// TIA Portal project "BTL_PLC_192" (V15)

(* hardware
DEVICE "S7300/ET200M station_1"  S7-300 station
   slot 0: "Rail_0"  Rail  6ES7 390-1***0-0AA0
   slot 2: "PLC_1"  CPU 314C-2 PN/DP  6ES7 314-6EH04-0AB0  V3.3
      slot 2: "PROFINET interface_1"  PN-IO
         slot 1: "Port_1"  Port
         slot 2: "Port_2"  Port
      slot 5: "DI 24/DO 16_1"  DI24/DO16
      slot 6: "AI 5/AO 2_1"  AI5/AO2
      slot 7: "Count_1"  Counter
      slot 8: "Positioning_1"  Positioning
*)

// ===== PLC "PLC_1"  CPU 314C-2 PN/DP =====

VAR_GLOBAL   // PLC tag table "Default tag table"
   "BI_AUTO" AT %I0.0 : Bool;
   "BI_MANU" AT %I0.1 : Bool;
   "BI_START" AT %I0.2 : Bool;
   "BI_STOP" AT %I0.3 : Bool;
   "I_CT1" AT %I0.4 : Bool;
   "I_CT2" AT %I0.5 : Bool;
   "I_CT3" AT %I0.6 : Bool;
   "I_CT4" AT %I0.7 : Bool;
   "IW_NHIET_DO" AT %IW64 : Int;
   "IW_ANH_SANG" AT %IW66 : Int;
   "IW_DO_AM" AT %IW68 : Int;
   "IW_DO_AM_DAT" AT %IW70 : Int;
   "BM_AUTO" AT %M0.0 : Bool;
   "BM_MANU" AT %M0.1 : Bool;
   "BM_START" AT %M0.2 : Bool;
   "BM_STOP" AT %M0.3 : Bool;
   "M_CT1" AT %M0.4 : Bool;
   "M_CT2" AT %M0.5 : Bool;
   "M_CT3" AT %M0.6 : Bool;
   "M_CT4" AT %M0.7 : Bool;
   "MW_NHIET_DO" AT %MW64 : Int;
   "MW_ANH_SANG" AT %MW66 : Int;
   "MW_DO_AM" AT %MW68 : Int;
   "MW_DO_AM_DAT" AT %MW70 : Int;
   "BM_SIMULATION" AT %M1.0 : Bool;
   "BIT_GIU" AT %M1.1 : Bool;
   "BIT_TUOI_THEO_TIME_THUC" AT %M1.2 : Bool;
   "BIT_TUOI_THEO_ND" AT %M1.3 : Bool;
   "BIT_TUOI_THEO_DA" AT %M1.4 : Bool;
   "BIT_TUOI_THEO_DAD" AT %M1.5 : Bool;
   "Q_DEN_LV" AT %Q0.0 : Bool;
   "Q_QTG1" AT %Q0.1 : Bool;
   "Q_QTG2" AT %Q0.2 : Bool;
   "Q_BPS" AT %Q0.3 : Bool;
   "Q_GN1" AT %Q0.4 : Bool;
   "Q_GN2" AT %Q0.5 : Bool;
   "Q_MC_CLOSE" AT %Q0.6 : Bool;
   "Q_MC_OPEN" AT %Q0.7 : Bool;
   "Q_BNV" AT %Q1.0 : Bool;
   "Q_QHA1" AT %Q1.1 : Bool;
   "Q_QHA2" AT %Q1.2 : Bool;
   "Q_DCS" AT %Q1.3 : Bool;
   "Auto" AT %M1.6 : Bool;
   "Manu" AT %M1.7 : Bool;
   "AUTO_RUN" AT %M2.0 : Bool;
   "MANU_RUN" AT %M2.1 : Bool;
   "SIM_MODE" AT %M2.2 : Bool;
   "RET_VAL1" AT %MW4 : Word;
   "BIPOLAR" AT %M2.3 : Bool;
   "RET_VAL2" AT %MW6 : Word;
   "RET_VAL3" AT %MW8 : Word;
   "RET_VAL4" AT %MW10 : Word;
   "RET_VAL5" AT %MW12 : Int;
   "ALWAY_OFF" AT %M2.4 : Bool;
   "TT_DATE_OF_WEEK" AT %MW194 : Int;
   "Tag_M" AT %M2.6 : Bool;
   "Tag_M1" AT %M2.7 : Bool;
   "TIME_TUOI" AT %MW14 : Int;
   "tag_M3" AT %M2.5 : Bool;
   "tag_M4" AT %M3.0 : Bool;
   "Tag_M5" AT %M3.1 : Bool;
   "Tag_M6" AT %M3.2 : Bool;
   "Tag_M7" AT %M3.3 : Bool;
   "Tag_M8" AT %M3.4 : Bool;
   "Tag_M9" AT %M3.5 : Bool;
   "Tag_1" AT %T1 : Timer;
END_VAR

VAR_GLOBAL   // PLC tag table "Tag table_1"
   "TT_NHIET_DO" AT %MD100 : Real;
   "TT_ANH_SANG" AT %MD104 : Real;
   "TT_DO_AM" AT %MD108 : Real;
   "SET_MAX_ND" AT %MD112 : Real;
   "SET_MIN_ND" AT %MD116 : Real;
   "SET_MAX_AS" AT %MD120 : Real;
   "SET_MIN_AS" AT %MD124 : Real;
   "SET_MAX_DO_AM" AT %MD128 : Real;
   "SET_MIN_DO_AM" AT %MD132 : Real;
   "SET_NGAY1" AT %MW148 : Int;
   "SET_GIO1" AT %MW150 : Int;
   "SET_PHUT1" AT %MW152 : Int;
   "TT_NGAY" AT %MW154 : Int;
   "TT_GIO" AT %MW156 : Int;
   "TT_PHUT" AT %MW158 : Int;
   "TT_GIAY" AT %MW160 : Int;
   "TT_NAM" AT %MW162 : Int;
   "TT_THANG" AT %MW164 : Int;
   "SET_NGAY2" AT %MW166 : Int;
   "SET_GIO2" AT %MW168 : Int;
   "SET_PHUT2" AT %MW170 : Int;
   "SET_NGAY3" AT %MW172 : Int;
   "SET_GIO3" AT %MW174 : Int;
   "SET_PHUT3" AT %MW176 : Int;
   "SET_TIME_TUOI" AT %MW178 : Int;
   "SET_MAX_DO_AM_DAT" AT %MD200 : Real;
   "SET_MIN_DO_AM_DAT" AT %MD204 : Real;
   "TT_DO_AM_DAT" AT %MD208 : Real;
   "TT_TIME_TUOI" AT %MW214 : Int;
   "SET_NHIET_DO" AT %MD216 : Real;
   "SET_DAD" AT %MD220 : Real;
   "SET_DO_AM_KK" AT %MD224 : Real;
   "SET_ANH_SANG" AT %MD228 : Real;
END_VAR

VAR_GLOBAL   // PLC tag table "Tag table_2"
   "START_BPS" AT %M20.0 : Bool;
   "STOP_BPS" AT %M20.1 : Bool;
   "START_QTG" AT %M20.2 : Bool;
   "STOP_QTG" AT %M20.3 : Bool;
   "START_DEN_CHIEU_SANG" AT %M20.4 : Bool;
   "STOP_DEN_CHIEU_SANG" AT %M20.5 : Bool;
   "START_QUAT_HUT_AM" AT %M20.6 : Bool;
   "STOP_QUAT_HUT_AM" AT %M20.7 : Bool;
   "START_GN" AT %M21.0 : Bool;
   "STOP_GN" AT %M21.1 : Bool;
   "OPEN_MAI_CHE" AT %M21.2 : Bool;
   "CLOSE_MAI_CHE" AT %M21.3 : Bool;
END_VAR

FUNCTION "MAY BOM SUONG" : Void   // FC1, LAD
{ S7_Optimized_Access := 'FALSE' }
VERSION : 0.1
   VAR_INPUT
      SET_GIO1 : Int;
      SET_PHUT1 : Int;
      SET_GIO2 : Int;
      SET_PHUT2 : Int;
      SET_GIO3 : Int;
      SET_PHUT3 : Int;
   END_VAR
   VAR_OUTPUT
      MAY_BOM_PS : Bool;
      GIA_NHIET1 : Bool;
      GIA_NHIET2 : Bool;
      QUAT_TG1 : Bool;
      QUAT_TG2 : Bool;
      QUAT_HUT_AM1 : Bool;
      QUAT_HUT_AM2 : Bool;
      BOM_NUOC_TANK : Bool;
   END_VAR
   VAR_TEMP
      ALWAYS_OFF : Bool;
      temp : Bool;
      LOOP : Bool;
      temp2 : Bool;
      TT_TUOI : Int;
   END_VAR
   VAR_TEMP   // added for the SCL form of the ladder/FBD networks
      _w1 : Bool;
   END_VAR
BEGIN

REGION Network 1: Đặt thời gian tưới trong ngày( tưới 3 lần 1 ngày)
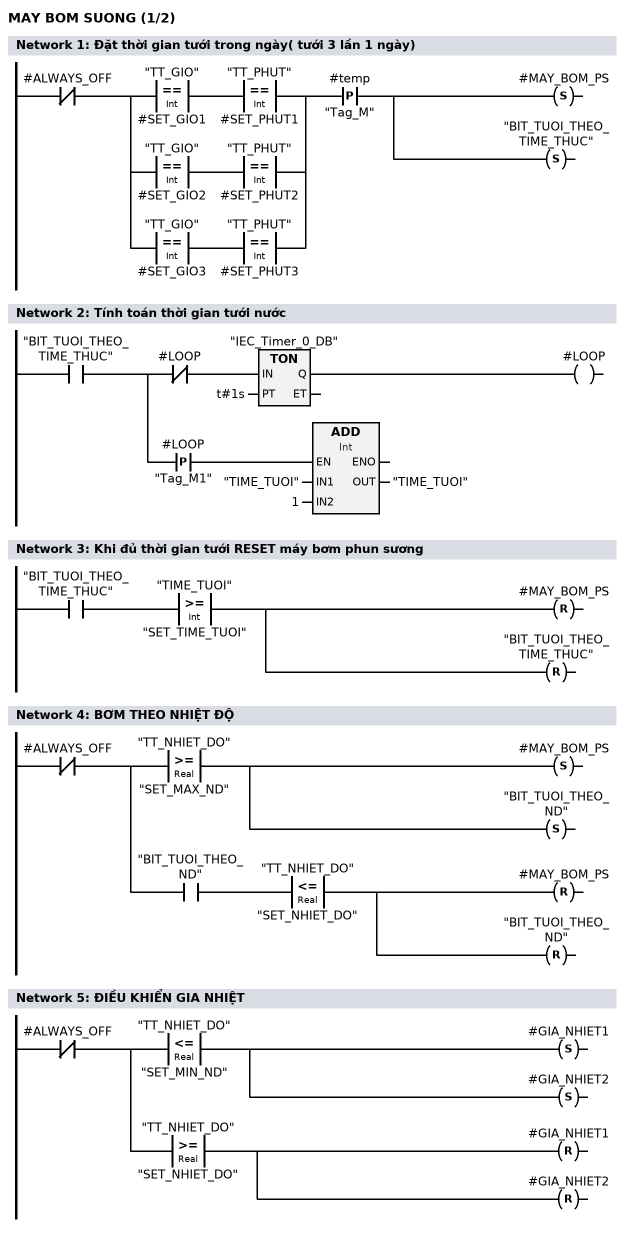
   RUNG wire#powerrail
      I_Contact( #ALWAYS_OFF )
      wire#w1
      { S7_Templates := "SrcType := Int" } EQ_Contact(in1 := "TT_GIO", in2 := #SET_GIO1)
      { S7_Templates := "SrcType := Int" } EQ_Contact(in1 := "TT_PHUT", in2 := #SET_PHUT1)
      wire#w2
      P_Contact(operand := #temp, bit := "Tag_M")
      wire#w3
      S_Coil( #MAY_BOM_PS )
   END_RUNG
   RUNG wire#w1
      { S7_Templates := "SrcType := Int" } EQ_Contact(in1 := "TT_GIO", in2 := #SET_GIO2)
      { S7_Templates := "SrcType := Int" } EQ_Contact(in1 := "TT_PHUT", in2 := #SET_PHUT2)
   END_RUNG wire#w2
   RUNG wire#w1
      { S7_Templates := "SrcType := Int" } EQ_Contact(in1 := "TT_GIO", in2 := #SET_GIO3)
      { S7_Templates := "SrcType := Int" } EQ_Contact(in1 := "TT_PHUT", in2 := #SET_PHUT3)
   END_RUNG wire#w2
   RUNG wire#w3
      S_Coil( "BIT_TUOI_THEO_TIME_THUC" )
   END_RUNG
   // the same network as SCL:
   #_w1 := NOT #ALWAYS_OFF AND ((("TT_GIO" = #SET_GIO1) AND ("TT_PHUT" = #SET_PHUT1)) OR (("TT_GIO" = #SET_GIO2) AND ("TT_PHUT" = #SET_PHUT2)) OR (("TT_GIO" = #SET_GIO3) AND ("TT_PHUT" = #SET_PHUT3))) AND #temp AND NOT "Tag_M";   // rising edge of #temp
   "Tag_M" := #temp;
   IF #_w1 THEN
       #MAY_BOM_PS := TRUE;
       "BIT_TUOI_THEO_TIME_THUC" := TRUE;
   END_IF;
END_REGION

REGION Network 2: Tính toán thời gian tưới nước
   "IEC_Timer_0_DB".TON(IN := "BIT_TUOI_THEO_TIME_THUC" AND NOT #LOOP, PT := t#1s);
   #LOOP := "IEC_Timer_0_DB".Q;
   #_w1 := "BIT_TUOI_THEO_TIME_THUC" AND #LOOP AND NOT "Tag_M1";   // rising edge of #LOOP
   "Tag_M1" := #LOOP;
   IF #_w1 THEN "TIME_TUOI" := "TIME_TUOI" + 1; END_IF;
END_REGION

REGION Network 3: Khi đủ thời gian tưới RESET máy bơm phun sương
   RUNG wire#powerrail
      Contact( "BIT_TUOI_THEO_TIME_THUC" )
      { S7_Templates := "SrcType := Int" } GE_Contact(in1 := "TIME_TUOI", in2 := "SET_TIME_TUOI")
      wire#w1
      R_Coil( #MAY_BOM_PS )
   END_RUNG
   RUNG wire#w1
      R_Coil( "BIT_TUOI_THEO_TIME_THUC" )
   END_RUNG
   // the same network as SCL:
   IF "BIT_TUOI_THEO_TIME_THUC" AND ("TIME_TUOI" >= "SET_TIME_TUOI") THEN
       #MAY_BOM_PS := FALSE;
       "BIT_TUOI_THEO_TIME_THUC" := FALSE;
   END_IF;
END_REGION

REGION Network 4: BƠM THEO NHIỆT ĐỘ
   RUNG wire#powerrail
      I_Contact( #ALWAYS_OFF )
      wire#w1
      { S7_Templates := "SrcType := Real" } GE_Contact(in1 := "TT_NHIET_DO", in2 := "SET_MAX_ND")
      wire#w2
      S_Coil( #MAY_BOM_PS )
   END_RUNG
   RUNG wire#w2
      S_Coil( "BIT_TUOI_THEO_ND" )
   END_RUNG
   RUNG wire#w1
      Contact( "BIT_TUOI_THEO_ND" )
      { S7_Templates := "SrcType := Real" } LE_Contact(in1 := "TT_NHIET_DO", in2 := "SET_NHIET_DO")
      wire#w3
      R_Coil( #MAY_BOM_PS )
   END_RUNG
   RUNG wire#w3
      R_Coil( "BIT_TUOI_THEO_ND" )
   END_RUNG
   // the same network as SCL:
   IF NOT #ALWAYS_OFF AND ("TT_NHIET_DO" >= "SET_MAX_ND") THEN
       #MAY_BOM_PS := TRUE;
       "BIT_TUOI_THEO_ND" := TRUE;
   END_IF;
   IF NOT #ALWAYS_OFF AND "BIT_TUOI_THEO_ND" AND ("TT_NHIET_DO" <= "SET_NHIET_DO") THEN
       #MAY_BOM_PS := FALSE;
       "BIT_TUOI_THEO_ND" := FALSE;
   END_IF;
END_REGION

REGION Network 5: ĐIỀU KHIỂN GIA NHIỆT
   RUNG wire#powerrail
      I_Contact( #ALWAYS_OFF )
      wire#w1
      { S7_Templates := "SrcType := Real" } LE_Contact(in1 := "TT_NHIET_DO", in2 := "SET_MIN_ND")
      wire#w2
      S_Coil( #GIA_NHIET1 )
   END_RUNG
   RUNG wire#w2
      S_Coil( #GIA_NHIET2 )
   END_RUNG
   RUNG wire#w1
      { S7_Templates := "SrcType := Real" } GE_Contact(in1 := "TT_NHIET_DO", in2 := "SET_NHIET_DO")
      wire#w3
      R_Coil( #GIA_NHIET1 )
   END_RUNG
   RUNG wire#w3
      R_Coil( #GIA_NHIET2 )
   END_RUNG
   // the same network as SCL:
   IF NOT #ALWAYS_OFF AND ("TT_NHIET_DO" <= "SET_MIN_ND") THEN
       #GIA_NHIET1 := TRUE;
       #GIA_NHIET2 := TRUE;
   END_IF;
   IF NOT #ALWAYS_OFF AND ("TT_NHIET_DO" >= "SET_NHIET_DO") THEN
       #GIA_NHIET1 := FALSE;
       #GIA_NHIET2 := FALSE;
   END_IF;
END_REGION

REGION Network 6: ĐIỀU KHIỂN MÁY BƠM THEO ĐỘ ẨM ĐẤT
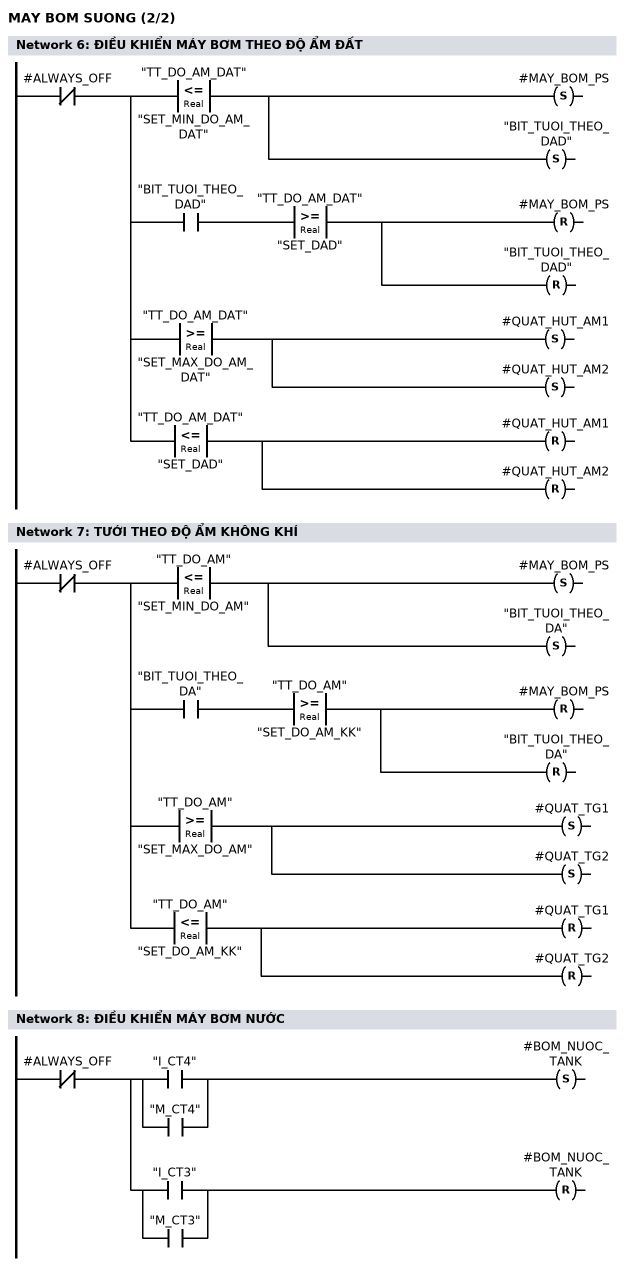
   RUNG wire#powerrail
      I_Contact( #ALWAYS_OFF )
      wire#w1
      { S7_Templates := "SrcType := Real" } LE_Contact(in1 := "TT_DO_AM_DAT", in2 := "SET_MIN_DO_AM_DAT")
      wire#w2
      S_Coil( #MAY_BOM_PS )
   END_RUNG
   RUNG wire#w2
      S_Coil( "BIT_TUOI_THEO_DAD" )
   END_RUNG
   RUNG wire#w1
      Contact( "BIT_TUOI_THEO_DAD" )
      { S7_Templates := "SrcType := Real" } GE_Contact(in1 := "TT_DO_AM_DAT", in2 := "SET_DAD")
      wire#w3
      R_Coil( #MAY_BOM_PS )
   END_RUNG
   RUNG wire#w3
      R_Coil( "BIT_TUOI_THEO_DAD" )
   END_RUNG
   RUNG wire#w1
      { S7_Templates := "SrcType := Real" } GE_Contact(in1 := "TT_DO_AM_DAT", in2 := "SET_MAX_DO_AM_DAT")
      wire#w4
      S_Coil( #QUAT_HUT_AM1 )
   END_RUNG
   RUNG wire#w4
      S_Coil( #QUAT_HUT_AM2 )
   END_RUNG
   RUNG wire#w1
      { S7_Templates := "SrcType := Real" } LE_Contact(in1 := "TT_DO_AM_DAT", in2 := "SET_DAD")
      wire#w5
      R_Coil( #QUAT_HUT_AM1 )
   END_RUNG
   RUNG wire#w5
      R_Coil( #QUAT_HUT_AM2 )
   END_RUNG
   // the same network as SCL:
   IF NOT #ALWAYS_OFF AND ("TT_DO_AM_DAT" <= "SET_MIN_DO_AM_DAT") THEN
       #MAY_BOM_PS := TRUE;
       "BIT_TUOI_THEO_DAD" := TRUE;
   END_IF;
   IF NOT #ALWAYS_OFF AND "BIT_TUOI_THEO_DAD" AND ("TT_DO_AM_DAT" >= "SET_DAD") THEN
       #MAY_BOM_PS := FALSE;
       "BIT_TUOI_THEO_DAD" := FALSE;
   END_IF;
   IF NOT #ALWAYS_OFF AND ("TT_DO_AM_DAT" >= "SET_MAX_DO_AM_DAT") THEN
       #QUAT_HUT_AM1 := TRUE;
       #QUAT_HUT_AM2 := TRUE;
   END_IF;
   IF NOT #ALWAYS_OFF AND ("TT_DO_AM_DAT" <= "SET_DAD") THEN
       #QUAT_HUT_AM1 := FALSE;
       #QUAT_HUT_AM2 := FALSE;
   END_IF;
END_REGION

REGION Network 7: TƯỚI THEO ĐỘ ẨM KHÔNG KHÍ
   RUNG wire#powerrail
      I_Contact( #ALWAYS_OFF )
      wire#w1
      { S7_Templates := "SrcType := Real" } LE_Contact(in1 := "TT_DO_AM", in2 := "SET_MIN_DO_AM")
      wire#w2
      S_Coil( #MAY_BOM_PS )
   END_RUNG
   RUNG wire#w2
      S_Coil( "BIT_TUOI_THEO_DA" )
   END_RUNG
   RUNG wire#w1
      Contact( "BIT_TUOI_THEO_DA" )
      { S7_Templates := "SrcType := Real" } GE_Contact(in1 := "TT_DO_AM", in2 := "SET_DO_AM_KK")
      wire#w3
      R_Coil( #MAY_BOM_PS )
   END_RUNG
   RUNG wire#w3
      R_Coil( "BIT_TUOI_THEO_DA" )
   END_RUNG
   RUNG wire#w1
      { S7_Templates := "SrcType := Real" } GE_Contact(in1 := "TT_DO_AM", in2 := "SET_MAX_DO_AM")
      wire#w4
      S_Coil( #QUAT_TG1 )
   END_RUNG
   RUNG wire#w4
      S_Coil( #QUAT_TG2 )
   END_RUNG
   RUNG wire#w1
      { S7_Templates := "SrcType := Real" } LE_Contact(in1 := "TT_DO_AM", in2 := "SET_DO_AM_KK")
      wire#w5
      R_Coil( #QUAT_TG1 )
   END_RUNG
   RUNG wire#w5
      R_Coil( #QUAT_TG2 )
   END_RUNG
   // the same network as SCL:
   IF NOT #ALWAYS_OFF AND ("TT_DO_AM" <= "SET_MIN_DO_AM") THEN
       #MAY_BOM_PS := TRUE;
       "BIT_TUOI_THEO_DA" := TRUE;
   END_IF;
   IF NOT #ALWAYS_OFF AND "BIT_TUOI_THEO_DA" AND ("TT_DO_AM" >= "SET_DO_AM_KK") THEN
       #MAY_BOM_PS := FALSE;
       "BIT_TUOI_THEO_DA" := FALSE;
   END_IF;
   IF NOT #ALWAYS_OFF AND ("TT_DO_AM" >= "SET_MAX_DO_AM") THEN
       #QUAT_TG1 := TRUE;
       #QUAT_TG2 := TRUE;
   END_IF;
   IF NOT #ALWAYS_OFF AND ("TT_DO_AM" <= "SET_DO_AM_KK") THEN
       #QUAT_TG1 := FALSE;
       #QUAT_TG2 := FALSE;
   END_IF;
END_REGION

REGION Network 8: ĐIỀU KHIỂN MÁY BƠM NƯỚC
   RUNG wire#powerrail
      I_Contact( #ALWAYS_OFF )
      wire#w1
      Contact( "I_CT4" )
      wire#w2
      S_Coil( #BOM_NUOC_TANK )
   END_RUNG
   RUNG wire#w1
      Contact( "M_CT4" )
   END_RUNG wire#w2
   RUNG wire#w1
      Contact( "I_CT3" )
      wire#w3
      R_Coil( #BOM_NUOC_TANK )
   END_RUNG
   RUNG wire#w1
      Contact( "M_CT3" )
   END_RUNG wire#w3
   // the same network as SCL:
   IF NOT #ALWAYS_OFF AND ("I_CT4" OR "M_CT4") THEN #BOM_NUOC_TANK := TRUE; END_IF;
   IF NOT #ALWAYS_OFF AND ("I_CT3" OR "M_CT3") THEN #BOM_NUOC_TANK := FALSE; END_IF;
END_REGION
END_FUNCTION

FUNCTION "MAI CHE" : Void   // FC2, LAD
{ S7_Optimized_Access := 'FALSE' }
VERSION : 0.1
   VAR_INPUT
      TT_ANH_SANG : Real;
      SET_MAX_AS : Real;
      SET_ANH_SANG : Real;
      SET_MIN_AS : Real;
   END_VAR
   VAR_OUTPUT
      MO_MAI_CHE : Bool;
      DEN_CHIEU_SANG : Bool;
      DONG_MAI_CHE : Bool;
   END_VAR
   VAR_TEMP
      ALWAYS_OFF : Bool;
   END_VAR
BEGIN

REGION Network 1
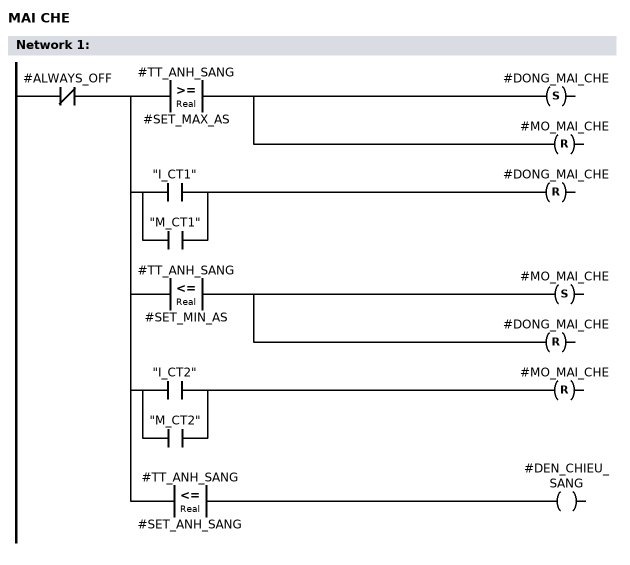
   RUNG wire#powerrail
      I_Contact( #ALWAYS_OFF )
      wire#w1
      { S7_Templates := "SrcType := Real" } GE_Contact(in1 := #TT_ANH_SANG, in2 := #SET_MAX_AS)
      wire#w2
      S_Coil( #DONG_MAI_CHE )
   END_RUNG
   RUNG wire#w2
      R_Coil( #MO_MAI_CHE )
   END_RUNG
   RUNG wire#w1
      Contact( "I_CT1" )
      wire#w3
      R_Coil( #DONG_MAI_CHE )
   END_RUNG
   RUNG wire#w1
      Contact( "M_CT1" )
   END_RUNG wire#w3
   RUNG wire#w1
      { S7_Templates := "SrcType := Real" } LE_Contact(in1 := #TT_ANH_SANG, in2 := #SET_MIN_AS)
      wire#w4
      S_Coil( #MO_MAI_CHE )
   END_RUNG
   RUNG wire#w4
      R_Coil( #DONG_MAI_CHE )
   END_RUNG
   RUNG wire#w1
      Contact( "I_CT2" )
      wire#w5
      R_Coil( #MO_MAI_CHE )
   END_RUNG
   RUNG wire#w1
      Contact( "M_CT2" )
   END_RUNG wire#w5
   RUNG wire#w1
      { S7_Templates := "SrcType := Real" } LE_Contact(in1 := #TT_ANH_SANG, in2 := #SET_ANH_SANG)
      Coil( #DEN_CHIEU_SANG )
   END_RUNG
   // the same network as SCL:
   IF NOT #ALWAYS_OFF AND (#TT_ANH_SANG >= #SET_MAX_AS) THEN
       #DONG_MAI_CHE := TRUE;
       #MO_MAI_CHE := FALSE;
   END_IF;
   IF NOT #ALWAYS_OFF AND ("I_CT1" OR "M_CT1") THEN #DONG_MAI_CHE := FALSE; END_IF;
   IF NOT #ALWAYS_OFF AND (#TT_ANH_SANG <= #SET_MIN_AS) THEN
       #MO_MAI_CHE := TRUE;
       #DONG_MAI_CHE := FALSE;
   END_IF;
   IF NOT #ALWAYS_OFF AND ("I_CT2" OR "M_CT2") THEN #MO_MAI_CHE := FALSE; END_IF;
   #DEN_CHIEU_SANG := NOT #ALWAYS_OFF AND (#TT_ANH_SANG <= #SET_ANH_SANG);
END_REGION
END_FUNCTION

FUNCTION "CHON CHE DO" : Void   // FC3, LAD
{ S7_Optimized_Access := 'FALSE' }
VERSION : 0.1
   VAR_INPUT
      S_AUTO : Bool;
      S_MANU : Bool;
      START : Bool;
      STOP : Bool;
   END_VAR
   VAR_OUTPUT
      MODE_AUTO : Bool;
      MODE_MANU : Bool;
   END_VAR
   VAR_TEMP
      AUTO : Bool;
      MANU : Bool;
   END_VAR
   VAR_TEMP   // added for the SCL form of the ladder/FBD networks
      _w1 : Bool;
   END_VAR
BEGIN

REGION Network 1
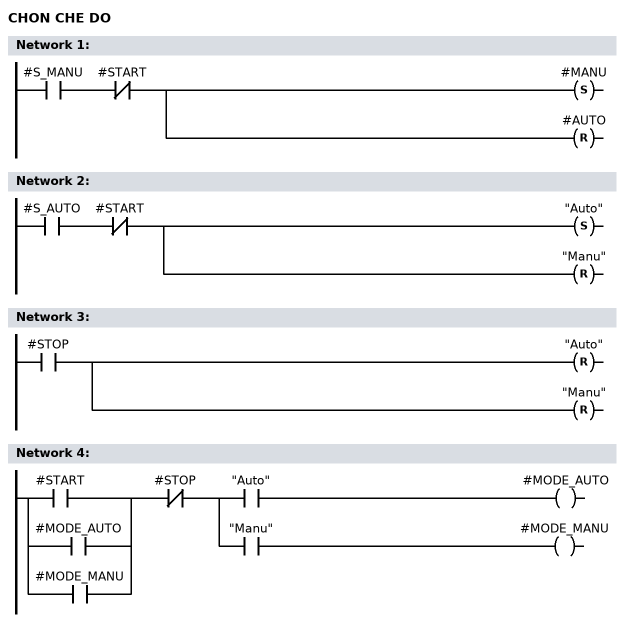
   RUNG wire#powerrail
      Contact( #S_MANU )
      I_Contact( #START )
      wire#w1
      S_Coil( #MANU )
   END_RUNG
   RUNG wire#w1
      R_Coil( #AUTO )
   END_RUNG
   // the same network as SCL:
   IF #S_MANU AND NOT #START THEN
       #MANU := TRUE;
       #AUTO := FALSE;
   END_IF;
END_REGION

REGION Network 2
   RUNG wire#powerrail
      Contact( #S_AUTO )
      I_Contact( #START )
      wire#w1
      S_Coil( "Auto" )
   END_RUNG
   RUNG wire#w1
      R_Coil( "Manu" )
   END_RUNG
   // the same network as SCL:
   IF #S_AUTO AND NOT #START THEN
       "Auto" := TRUE;
       "Manu" := FALSE;
   END_IF;
END_REGION

REGION Network 3
   RUNG wire#powerrail
      Contact( #STOP )
      wire#w1
      R_Coil( "Auto" )
   END_RUNG
   RUNG wire#w1
      R_Coil( "Manu" )
   END_RUNG
   // the same network as SCL:
   IF #STOP THEN
       "Auto" := FALSE;
       "Manu" := FALSE;
   END_IF;
END_REGION

REGION Network 4
   RUNG wire#powerrail
      Contact( #START )
      wire#w1
      I_Contact( #STOP )
      wire#w2
      Contact( "Auto" )
      Coil( #MODE_AUTO )
   END_RUNG
   RUNG wire#powerrail
      Contact( #MODE_AUTO )
   END_RUNG wire#w1
   RUNG wire#powerrail
      Contact( #MODE_MANU )
   END_RUNG wire#w1
   RUNG wire#w2
      Contact( "Manu" )
      Coil( #MODE_MANU )
   END_RUNG
   // the same network as SCL:
   #_w1 := (#START OR #MODE_AUTO OR #MODE_MANU) AND NOT #STOP;
   #MODE_AUTO := #_w1 AND "Auto";
   #MODE_MANU := #_w1 AND "Manu";
END_REGION
END_FUNCTION

FUNCTION "CONDITION" : Void   // FC4, LAD
{ S7_Optimized_Access := 'FALSE' }
VERSION : 0.1
   VAR_INPUT
      SIM_MODE : Bool;
      MW_ANH_SANG : Int;
      MW_DO_AM : Int;
      MW_NHIET_DO : Int;
      MW_DO_AM_DAT : Int;
   END_VAR
   VAR_OUTPUT
      IW_ANH_SANG : Int;
      IW_DO_AM : Int;
      IW_NHIET_DO : Int;
      IW_DO_AM_DAT : Int;
   END_VAR
BEGIN

REGION Network 1
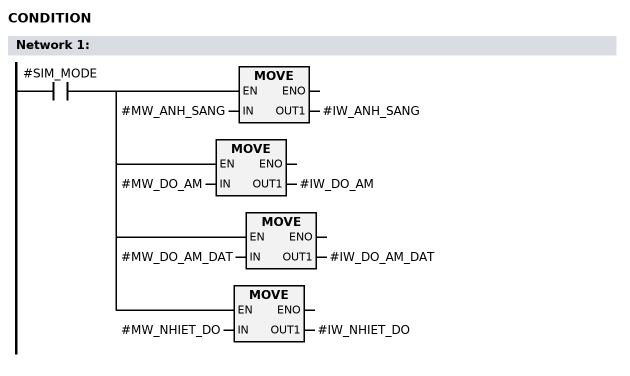
   RUNG wire#powerrail
      Contact( #SIM_MODE )
      wire#w1
      { S7_GenerateENO := "TRUE" } Move(in := #MW_ANH_SANG, out1 => #IW_ANH_SANG)
   END_RUNG
   RUNG wire#w1
      { S7_GenerateENO := "TRUE" } Move(in := #MW_DO_AM, out1 => #IW_DO_AM)
   END_RUNG
   RUNG wire#w1
      { S7_GenerateENO := "TRUE" } Move(in := #MW_DO_AM_DAT, out1 => #IW_DO_AM_DAT)
   END_RUNG
   RUNG wire#w1
      { S7_GenerateENO := "TRUE" } Move(in := #MW_NHIET_DO, out1 => #IW_NHIET_DO)
   END_RUNG
   // the same network as SCL:
   IF #SIM_MODE THEN
       #IW_ANH_SANG := #MW_ANH_SANG;
       #IW_DO_AM := #MW_DO_AM;
       #IW_DO_AM_DAT := #MW_DO_AM_DAT;
       #IW_NHIET_DO := #MW_NHIET_DO;
   END_IF;
END_REGION
END_FUNCTION

FUNCTION "MODE_MANUAL" : Void   // FC5, LAD
{ S7_Optimized_Access := 'FALSE' }
VERSION : 0.1
   VAR_INPUT
      START_BPS : Bool;
      STOP_BPS : Bool;
      START_QTG : Bool;
      STOP_QTG : Bool;
      START_DEN_CHIEU_SANG : Bool;
      STOP_DEN_CHIEU_SANG : Bool;
      START_QUAT_HUT_AM : Bool;
      STOP_QUAT_HUT_AM : Bool;
      START_GN : Bool;
      STOP_GN : Bool;
      OPEN_MAI_CHE : Bool;
      CLOSE_MAI_CHE : Bool;
   END_VAR
   VAR_OUTPUT
      BOM_NUOC_TANK : Bool;
      BOM_PHUN_SUONG : Bool;
      QUAT_TG1 : Bool;
      QUAT_TG2 : Bool;
      MAI_CHE_DONG : Bool;
      MAI_CHE_MO : Bool;
      DEN_CHIEU_SANG : Bool;
      QUAT_HUT_AM1 : Bool;
      QUAT_HUT_AM2 : Bool;
      GIA_NHIET1 : Bool;
      GIA_NHIET2 : Bool;
   END_VAR
   VAR_TEMP
      ALWAYS_OFF : Bool;
   END_VAR
BEGIN

REGION Network 1: ĐIỀU KHIỂN MÁY BƠM NƯỚC VÀO BỂ CHỨA
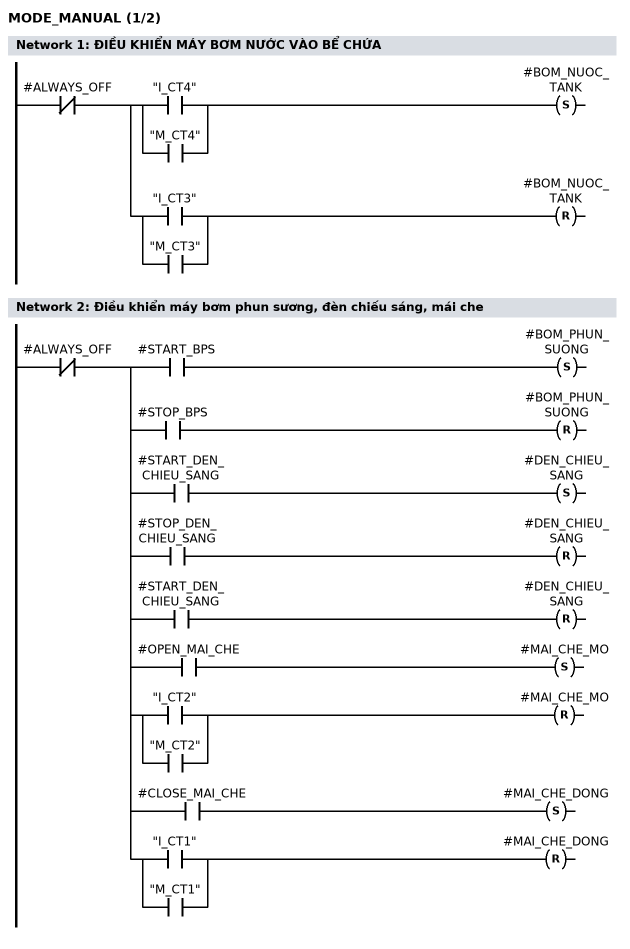
   RUNG wire#powerrail
      I_Contact( #ALWAYS_OFF )
      wire#w1
      Contact( "I_CT4" )
      wire#w2
      S_Coil( #BOM_NUOC_TANK )
   END_RUNG
   RUNG wire#w1
      Contact( "M_CT4" )
   END_RUNG wire#w2
   RUNG wire#w1
      Contact( "I_CT3" )
      wire#w3
      R_Coil( #BOM_NUOC_TANK )
   END_RUNG
   RUNG wire#w1
      Contact( "M_CT3" )
   END_RUNG wire#w3
   // the same network as SCL:
   IF NOT #ALWAYS_OFF AND ("I_CT4" OR "M_CT4") THEN #BOM_NUOC_TANK := TRUE; END_IF;
   IF NOT #ALWAYS_OFF AND ("I_CT3" OR "M_CT3") THEN #BOM_NUOC_TANK := FALSE; END_IF;
END_REGION

REGION Network 2: Điều khiển máy bơm phun sương, đèn chiếu sáng, mái che
   RUNG wire#powerrail
      I_Contact( #ALWAYS_OFF )
      wire#w1
      Contact( #START_BPS )
      S_Coil( #BOM_PHUN_SUONG )
   END_RUNG
   RUNG wire#w1
      Contact( #STOP_BPS )
      R_Coil( #BOM_PHUN_SUONG )
   END_RUNG
   RUNG wire#w1
      Contact( #START_DEN_CHIEU_SANG )
      S_Coil( #DEN_CHIEU_SANG )
   END_RUNG
   RUNG wire#w1
      Contact( #STOP_DEN_CHIEU_SANG )
      R_Coil( #DEN_CHIEU_SANG )
   END_RUNG
   RUNG wire#w1
      Contact( #START_DEN_CHIEU_SANG )
      R_Coil( #DEN_CHIEU_SANG )
   END_RUNG
   RUNG wire#w1
      Contact( #OPEN_MAI_CHE )
      S_Coil( #MAI_CHE_MO )
   END_RUNG
   RUNG wire#w1
      Contact( "I_CT2" )
      wire#w2
      R_Coil( #MAI_CHE_MO )
   END_RUNG
   RUNG wire#w1
      Contact( "M_CT2" )
   END_RUNG wire#w2
   RUNG wire#w1
      Contact( #CLOSE_MAI_CHE )
      S_Coil( #MAI_CHE_DONG )
   END_RUNG
   RUNG wire#w1
      Contact( "I_CT1" )
      wire#w3
      R_Coil( #MAI_CHE_DONG )
   END_RUNG
   RUNG wire#w1
      Contact( "M_CT1" )
   END_RUNG wire#w3
   // the same network as SCL:
   IF NOT #ALWAYS_OFF AND #START_BPS THEN #BOM_PHUN_SUONG := TRUE; END_IF;
   IF NOT #ALWAYS_OFF AND #STOP_BPS THEN #BOM_PHUN_SUONG := FALSE; END_IF;
   IF NOT #ALWAYS_OFF AND #START_DEN_CHIEU_SANG THEN #DEN_CHIEU_SANG := TRUE; END_IF;
   IF NOT #ALWAYS_OFF AND #STOP_DEN_CHIEU_SANG THEN #DEN_CHIEU_SANG := FALSE; END_IF;
   IF NOT #ALWAYS_OFF AND #START_DEN_CHIEU_SANG THEN #DEN_CHIEU_SANG := FALSE; END_IF;
   IF NOT #ALWAYS_OFF AND #OPEN_MAI_CHE THEN #MAI_CHE_MO := TRUE; END_IF;
   IF NOT #ALWAYS_OFF AND ("I_CT2" OR "M_CT2") THEN #MAI_CHE_MO := FALSE; END_IF;
   IF NOT #ALWAYS_OFF AND #CLOSE_MAI_CHE THEN #MAI_CHE_DONG := TRUE; END_IF;
   IF NOT #ALWAYS_OFF AND ("I_CT1" OR "M_CT1") THEN #MAI_CHE_DONG := FALSE; END_IF;
END_REGION

REGION Network 3: Quạt thông gió, quạt hút ẩm, gia nhiệt
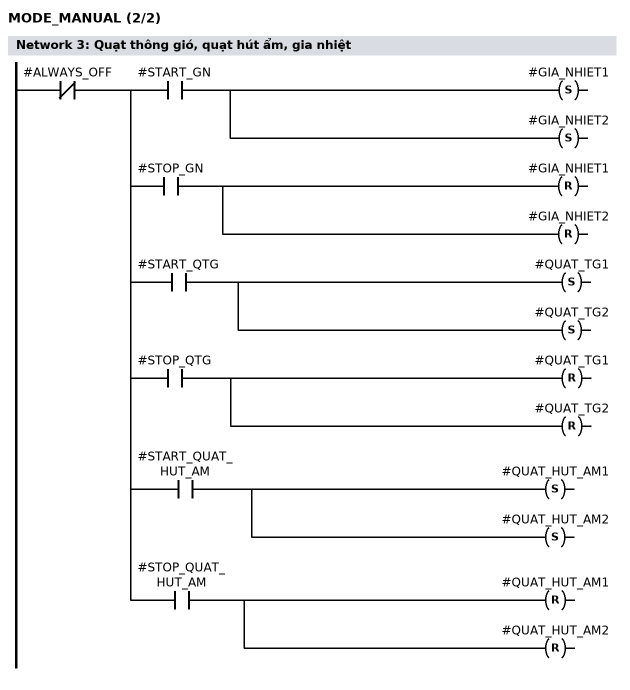
   RUNG wire#powerrail
      I_Contact( #ALWAYS_OFF )
      wire#w1
      Contact( #START_GN )
      wire#w2
      S_Coil( #GIA_NHIET1 )
   END_RUNG
   RUNG wire#w2
      S_Coil( #GIA_NHIET2 )
   END_RUNG
   RUNG wire#w1
      Contact( #STOP_GN )
      wire#w3
      R_Coil( #GIA_NHIET1 )
   END_RUNG
   RUNG wire#w3
      R_Coil( #GIA_NHIET2 )
   END_RUNG
   RUNG wire#w1
      Contact( #START_QTG )
      wire#w4
      S_Coil( #QUAT_TG1 )
   END_RUNG
   RUNG wire#w4
      S_Coil( #QUAT_TG2 )
   END_RUNG
   RUNG wire#w1
      Contact( #STOP_QTG )
      wire#w5
      R_Coil( #QUAT_TG1 )
   END_RUNG
   RUNG wire#w5
      R_Coil( #QUAT_TG2 )
   END_RUNG
   RUNG wire#w1
      Contact( #START_QUAT_HUT_AM )
      wire#w6
      S_Coil( #QUAT_HUT_AM1 )
   END_RUNG
   RUNG wire#w6
      S_Coil( #QUAT_HUT_AM2 )
   END_RUNG
   RUNG wire#w1
      Contact( #STOP_QUAT_HUT_AM )
      wire#w7
      R_Coil( #QUAT_HUT_AM1 )
   END_RUNG
   RUNG wire#w7
      R_Coil( #QUAT_HUT_AM2 )
   END_RUNG
   // the same network as SCL:
   IF NOT #ALWAYS_OFF AND #START_GN THEN
       #GIA_NHIET1 := TRUE;
       #GIA_NHIET2 := TRUE;
   END_IF;
   IF NOT #ALWAYS_OFF AND #STOP_GN THEN
       #GIA_NHIET1 := FALSE;
       #GIA_NHIET2 := FALSE;
   END_IF;
   IF NOT #ALWAYS_OFF AND #START_QTG THEN
       #QUAT_TG1 := TRUE;
       #QUAT_TG2 := TRUE;
   END_IF;
   IF NOT #ALWAYS_OFF AND #STOP_QTG THEN
       #QUAT_TG1 := FALSE;
       #QUAT_TG2 := FALSE;
   END_IF;
   IF NOT #ALWAYS_OFF AND #START_QUAT_HUT_AM THEN
       #QUAT_HUT_AM1 := TRUE;
       #QUAT_HUT_AM2 := TRUE;
   END_IF;
   IF NOT #ALWAYS_OFF AND #STOP_QUAT_HUT_AM THEN
       #QUAT_HUT_AM1 := FALSE;
       #QUAT_HUT_AM2 := FALSE;
   END_IF;
END_REGION
END_FUNCTION

FUNCTION "SIMULATE" : Void   // FC6, LAD
{ S7_Optimized_Access := 'FALSE' }
VERSION : 0.1
   VAR_TEMP
      LOOP : Bool;
      ALWAYS_OFF : Bool;
      temp2 : Bool;
   END_VAR
   VAR_TEMP   // added for the SCL form of the ladder/FBD networks
      _w1 : Bool;
      _w2 : Bool;
      _s5time1 : S5Time;
      _w3 : Bool;
      _w4 : Bool;
   END_VAR
BEGIN

REGION Network 1: CÔNG TẮC MÁI CHE
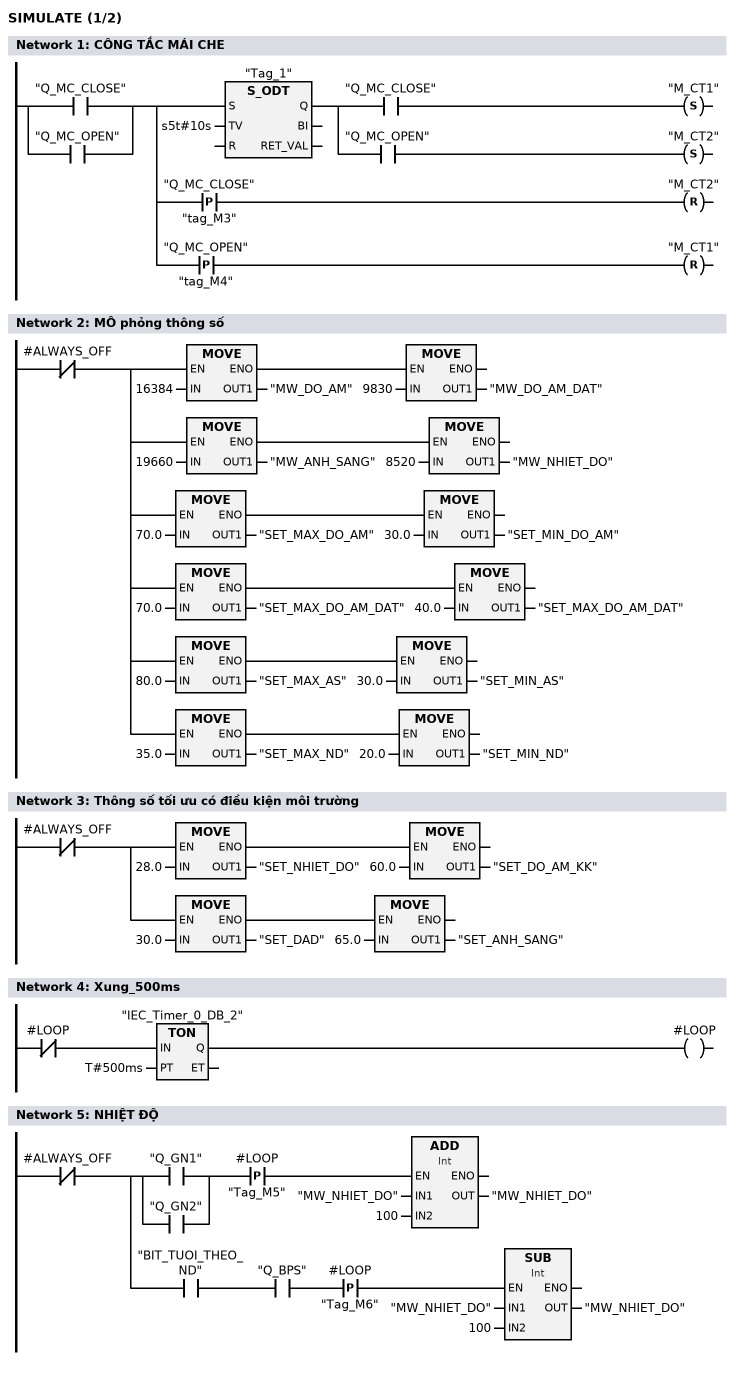
   RUNG wire#powerrail
      Contact( "Q_MC_CLOSE" )
      wire#w1
      S_ODT(T_NO := "Tag_1", TV := s5t#10s, R :=, BI =>, RET_VAL =>)
      wire#w2
      Contact( "Q_MC_CLOSE" )
      S_Coil( "M_CT1" )
   END_RUNG
   RUNG wire#powerrail
      Contact( "Q_MC_OPEN" )
   END_RUNG wire#w1
   RUNG wire#w2
      Contact( "Q_MC_OPEN" )
      S_Coil( "M_CT2" )
   END_RUNG
   RUNG wire#w1
      P_Contact(operand := "Q_MC_CLOSE", bit := "tag_M3")
      R_Coil( "M_CT2" )
   END_RUNG
   RUNG wire#w1
      P_Contact(operand := "Q_MC_OPEN", bit := "tag_M4")
      R_Coil( "M_CT1" )
   END_RUNG
   // the same network as SCL:
   #_w1 := "Q_MC_CLOSE" OR "Q_MC_OPEN";
   #_s5time1 := S_ODT(T_NO := "Tag_1", S := #_w1, TV := s5t#10s, Q => #_w2);
   IF #_w2 AND "Q_MC_CLOSE" THEN "M_CT1" := TRUE; END_IF;
   IF #_w2 AND "Q_MC_OPEN" THEN "M_CT2" := TRUE; END_IF;
   #_w3 := #_w1 AND "Q_MC_CLOSE" AND NOT "tag_M3";   // rising edge of "Q_MC_CLOSE"
   "tag_M3" := "Q_MC_CLOSE";
   IF #_w3 THEN "M_CT2" := FALSE; END_IF;
   #_w4 := #_w1 AND "Q_MC_OPEN" AND NOT "tag_M4";   // rising edge of "Q_MC_OPEN"
   "tag_M4" := "Q_MC_OPEN";
   IF #_w4 THEN "M_CT1" := FALSE; END_IF;
END_REGION

REGION Network 2: MÔ phỏng thông số
   RUNG wire#powerrail
      I_Contact( #ALWAYS_OFF )
      wire#w1
      { S7_GenerateENO := "TRUE" } Move(in := 16384, out1 => "MW_DO_AM")
      { S7_GenerateENO := "TRUE" } Move(in := 9830, out1 => "MW_DO_AM_DAT")
   END_RUNG
   RUNG wire#w1
      { S7_GenerateENO := "TRUE" } Move(in := 19660, out1 => "MW_ANH_SANG")
      { S7_GenerateENO := "TRUE" } Move(in := 8520, out1 => "MW_NHIET_DO")
   END_RUNG
   RUNG wire#w1
      { S7_GenerateENO := "TRUE" } Move(in := 70.0, out1 => "SET_MAX_DO_AM")
      { S7_GenerateENO := "TRUE" } Move(in := 30.0, out1 => "SET_MIN_DO_AM")
   END_RUNG
   RUNG wire#w1
      { S7_GenerateENO := "TRUE" } Move(in := 70.0, out1 => "SET_MAX_DO_AM_DAT")
      { S7_GenerateENO := "TRUE" } Move(in := 40.0, out1 => "SET_MAX_DO_AM_DAT")
   END_RUNG
   RUNG wire#w1
      { S7_GenerateENO := "TRUE" } Move(in := 80.0, out1 => "SET_MAX_AS")
      { S7_GenerateENO := "TRUE" } Move(in := 30.0, out1 => "SET_MIN_AS")
   END_RUNG
   RUNG wire#w1
      { S7_GenerateENO := "TRUE" } Move(in := 35.0, out1 => "SET_MAX_ND")
      { S7_GenerateENO := "TRUE" } Move(in := 20.0, out1 => "SET_MIN_ND")
   END_RUNG
   // the same network as SCL:
   // ENO of a box is taken as its EN; it also drops when the box reports an error
   IF NOT #ALWAYS_OFF THEN
       "MW_DO_AM" := 16384;
       "MW_DO_AM_DAT" := 9830;
       "MW_ANH_SANG" := 19660;
       "MW_NHIET_DO" := 8520;
       "SET_MAX_DO_AM" := 70.0;
       "SET_MIN_DO_AM" := 30.0;
       "SET_MAX_DO_AM_DAT" := 70.0;
       "SET_MAX_DO_AM_DAT" := 40.0;
       "SET_MAX_AS" := 80.0;
       "SET_MIN_AS" := 30.0;
       "SET_MAX_ND" := 35.0;
       "SET_MIN_ND" := 20.0;
   END_IF;
END_REGION

REGION Network 3: Thông số tối ưu có điều kiện môi trường
   RUNG wire#powerrail
      I_Contact( #ALWAYS_OFF )
      wire#w1
      { S7_GenerateENO := "TRUE" } Move(in := 28.0, out1 => "SET_NHIET_DO")
      { S7_GenerateENO := "TRUE" } Move(in := 60.0, out1 => "SET_DO_AM_KK")
   END_RUNG
   RUNG wire#w1
      { S7_GenerateENO := "TRUE" } Move(in := 30.0, out1 => "SET_DAD")
      { S7_GenerateENO := "TRUE" } Move(in := 65.0, out1 => "SET_ANH_SANG")
   END_RUNG
   // the same network as SCL:
   // ENO of a box is taken as its EN; it also drops when the box reports an error
   IF NOT #ALWAYS_OFF THEN
       "SET_NHIET_DO" := 28.0;
       "SET_DO_AM_KK" := 60.0;
       "SET_DAD" := 30.0;
       "SET_ANH_SANG" := 65.0;
   END_IF;
END_REGION

REGION Network 4: Xung_500ms
   "IEC_Timer_0_DB_2".TON(IN := NOT #LOOP, PT := T#500ms);
   #LOOP := "IEC_Timer_0_DB_2".Q;
END_REGION

REGION Network 5: NHIỆT ĐỘ
   RUNG wire#powerrail
      I_Contact( #ALWAYS_OFF )
      wire#w1
      Contact( "Q_GN1" )
      wire#w2
      P_Contact(operand := #LOOP, bit := "Tag_M5")
      { S7_Templates := "SrcType := Int"; S7_GenerateENO := "TRUE" } Add(in1 := "MW_NHIET_DO", in2 := 100, out => "MW_NHIET_DO")
   END_RUNG
   RUNG wire#w1
      Contact( "Q_GN2" )
   END_RUNG wire#w2
   RUNG wire#w1
      Contact( "BIT_TUOI_THEO_ND" )
      Contact( "Q_BPS" )
      P_Contact(operand := #LOOP, bit := "Tag_M6")
      { S7_Templates := "SrcType := Int"; S7_GenerateENO := "TRUE" } Sub(in1 := "MW_NHIET_DO", in2 := 100, out => "MW_NHIET_DO")
   END_RUNG
   // the same network as SCL:
   #_w1 := NOT #ALWAYS_OFF AND ("Q_GN1" OR "Q_GN2") AND #LOOP AND NOT "Tag_M5";   // rising edge of #LOOP
   "Tag_M5" := #LOOP;
   IF #_w1 THEN "MW_NHIET_DO" := "MW_NHIET_DO" + 100; END_IF;
   #_w2 := NOT #ALWAYS_OFF AND "BIT_TUOI_THEO_ND" AND "Q_BPS" AND #LOOP AND NOT "Tag_M6";   // rising edge of #LOOP
   "Tag_M6" := #LOOP;
   IF #_w2 THEN "MW_NHIET_DO" := "MW_NHIET_DO" - 100; END_IF;
END_REGION

REGION Network 6: ÁNH SÁNG
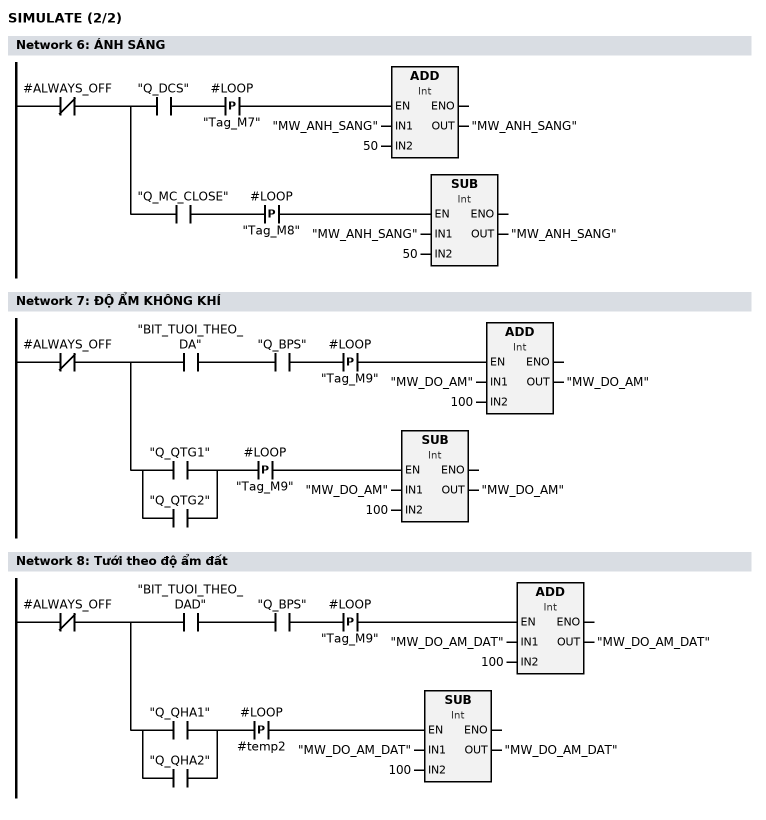
   RUNG wire#powerrail
      I_Contact( #ALWAYS_OFF )
      wire#w1
      Contact( "Q_DCS" )
      P_Contact(operand := #LOOP, bit := "Tag_M7")
      { S7_Templates := "SrcType := Int"; S7_GenerateENO := "TRUE" } Add(in1 := "MW_ANH_SANG", in2 := 50, out => "MW_ANH_SANG")
   END_RUNG
   RUNG wire#w1
      Contact( "Q_MC_CLOSE" )
      P_Contact(operand := #LOOP, bit := "Tag_M8")
      { S7_Templates := "SrcType := Int"; S7_GenerateENO := "TRUE" } Sub(in1 := "MW_ANH_SANG", in2 := 50, out => "MW_ANH_SANG")
   END_RUNG
   // the same network as SCL:
   #_w1 := NOT #ALWAYS_OFF AND "Q_DCS" AND #LOOP AND NOT "Tag_M7";   // rising edge of #LOOP
   "Tag_M7" := #LOOP;
   IF #_w1 THEN "MW_ANH_SANG" := "MW_ANH_SANG" + 50; END_IF;
   #_w2 := NOT #ALWAYS_OFF AND "Q_MC_CLOSE" AND #LOOP AND NOT "Tag_M8";   // rising edge of #LOOP
   "Tag_M8" := #LOOP;
   IF #_w2 THEN "MW_ANH_SANG" := "MW_ANH_SANG" - 50; END_IF;
END_REGION

REGION Network 7: ĐỘ ẨM KHÔNG KHÍ
   RUNG wire#powerrail
      I_Contact( #ALWAYS_OFF )
      wire#w1
      Contact( "BIT_TUOI_THEO_DA" )
      Contact( "Q_BPS" )
      P_Contact(operand := #LOOP, bit := "Tag_M9")
      { S7_Templates := "SrcType := Int"; S7_GenerateENO := "TRUE" } Add(in1 := "MW_DO_AM", in2 := 100, out => "MW_DO_AM")
   END_RUNG
   RUNG wire#w1
      Contact( "Q_QTG1" )
      wire#w2
      P_Contact(operand := #LOOP, bit := "Tag_M9")
      { S7_Templates := "SrcType := Int"; S7_GenerateENO := "TRUE" } Sub(in1 := "MW_DO_AM", in2 := 100, out => "MW_DO_AM")
   END_RUNG
   RUNG wire#w1
      Contact( "Q_QTG2" )
   END_RUNG wire#w2
   // the same network as SCL:
   #_w1 := NOT #ALWAYS_OFF AND "BIT_TUOI_THEO_DA" AND "Q_BPS" AND #LOOP AND NOT "Tag_M9";   // rising edge of #LOOP
   "Tag_M9" := #LOOP;
   IF #_w1 THEN "MW_DO_AM" := "MW_DO_AM" + 100; END_IF;
   #_w2 := NOT #ALWAYS_OFF AND ("Q_QTG1" OR "Q_QTG2") AND #LOOP AND NOT "Tag_M9";   // rising edge of #LOOP
   "Tag_M9" := #LOOP;
   IF #_w2 THEN "MW_DO_AM" := "MW_DO_AM" - 100; END_IF;
END_REGION

REGION Network 8: Tưới theo độ ẩm đất
   RUNG wire#powerrail
      I_Contact( #ALWAYS_OFF )
      wire#w1
      Contact( "BIT_TUOI_THEO_DAD" )
      Contact( "Q_BPS" )
      P_Contact(operand := #LOOP, bit := "Tag_M9")
      { S7_Templates := "SrcType := Int"; S7_GenerateENO := "TRUE" } Add(in1 := "MW_DO_AM_DAT", in2 := 100, out => "MW_DO_AM_DAT")
   END_RUNG
   RUNG wire#w1
      Contact( "Q_QHA1" )
      wire#w2
      P_Contact(operand := #LOOP, bit := #temp2)
      { S7_Templates := "SrcType := Int"; S7_GenerateENO := "TRUE" } Sub(in1 := "MW_DO_AM_DAT", in2 := 100, out => "MW_DO_AM_DAT")
   END_RUNG
   RUNG wire#w1
      Contact( "Q_QHA2" )
   END_RUNG wire#w2
   // the same network as SCL:
   #_w1 := NOT #ALWAYS_OFF AND "BIT_TUOI_THEO_DAD" AND "Q_BPS" AND #LOOP AND NOT "Tag_M9";   // rising edge of #LOOP
   "Tag_M9" := #LOOP;
   IF #_w1 THEN "MW_DO_AM_DAT" := "MW_DO_AM_DAT" + 100; END_IF;
   #_w2 := NOT #ALWAYS_OFF AND ("Q_QHA1" OR "Q_QHA2") AND #LOOP AND NOT #temp2;   // rising edge of #LOOP
   #temp2 := #LOOP;
   IF #_w2 THEN "MW_DO_AM_DAT" := "MW_DO_AM_DAT" - 100; END_IF;
END_REGION
END_FUNCTION

ORGANIZATION_BLOCK "Main"   // OB1, LAD
TITLE = "Main Program Sweep (Cycle)"
{ S7_Optimized_Access := 'FALSE' }
VERSION : 0.1
   VAR_TEMP
      OB1_EV_CLASS : Byte;   // Bits 0-3 = 1 (Coming event), Bits 4-7 = 1 (Event class 1)
      OB1_SCAN_1 : Byte;   // 1 (Cold restart scan 1 of OB 1), 3 (Scan 2-n of OB 1)
      OB1_PRIORITY : Byte;   // Priority of OB Execution
      OB1_OB_NUMBR : Byte;   // 1 (Organization block 1, OB1)
      OB1_RESERVED_1 : Byte;   // Reserved for system
      OB1_RESERVED_2 : Byte;   // Reserved for system
      OB1_PREV_CYCLE : Int;   // Cycle time of previous OB1 scan (milliseconds)
      OB1_MIN_CYCLE : Int;   // Minimum cycle time of OB1 (milliseconds)
      OB1_MAX_CYCLE : Int;   // Maximum cycle time of OB1 (milliseconds)
      OB1_DATE_TIME : Date_And_Time;   // Date and time OB1 started
   END_VAR
BEGIN

REGION Network 1: chọn mode manual hoặc auto
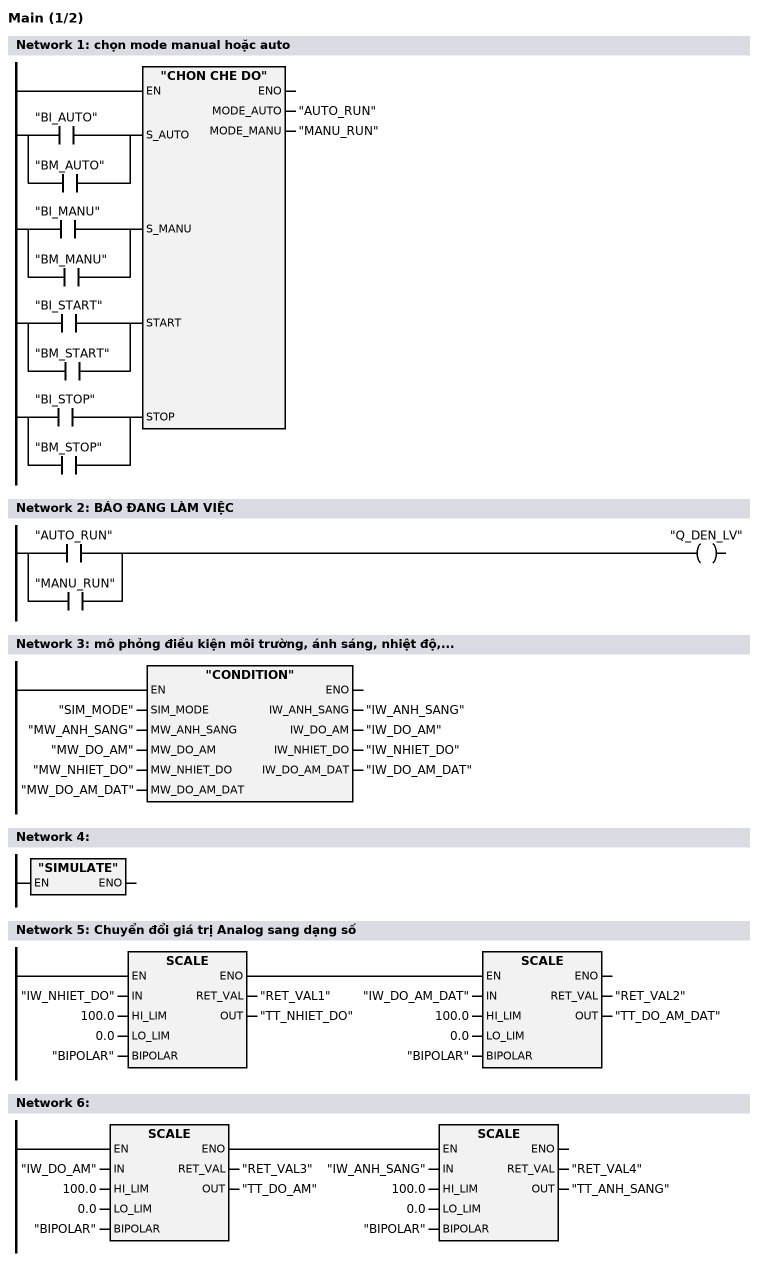
   RUNG wire#powerrail
      "CHON CHE DO"(S_AUTO := wire#w1, S_MANU := wire#w2, START := wire#w3, STOP := wire#w4, MODE_AUTO => "AUTO_RUN", MODE_MANU => "MANU_RUN")
   END_RUNG
   RUNG wire#powerrail
      Contact( "BI_AUTO" )
   END_RUNG wire#w1
   RUNG wire#powerrail
      Contact( "BM_AUTO" )
   END_RUNG wire#w1
   RUNG wire#powerrail
      Contact( "BI_MANU" )
   END_RUNG wire#w2
   RUNG wire#powerrail
      Contact( "BM_MANU" )
   END_RUNG wire#w2
   RUNG wire#powerrail
      Contact( "BI_START" )
   END_RUNG wire#w3
   RUNG wire#powerrail
      Contact( "BM_START" )
   END_RUNG wire#w3
   RUNG wire#powerrail
      Contact( "BI_STOP" )
   END_RUNG wire#w4
   RUNG wire#powerrail
      Contact( "BM_STOP" )
   END_RUNG wire#w4
   // the same network as SCL:
   "CHON CHE DO"(S_AUTO := "BI_AUTO" OR "BM_AUTO",
                 S_MANU := "BI_MANU" OR "BM_MANU",
                 START := "BI_START" OR "BM_START",
                 STOP := "BI_STOP" OR "BM_STOP",
                 MODE_AUTO => "AUTO_RUN",
                 MODE_MANU => "MANU_RUN");
END_REGION

REGION Network 2: BÁO ĐANG LÀM VIỆC
   RUNG wire#powerrail
      Contact( "AUTO_RUN" )
      wire#w1
      Coil( "Q_DEN_LV" )
   END_RUNG
   RUNG wire#powerrail
      Contact( "MANU_RUN" )
   END_RUNG wire#w1
   // the same network as SCL:
   "Q_DEN_LV" := "AUTO_RUN" OR "MANU_RUN";
END_REGION

REGION Network 3: mô phỏng điều kiện môi trường, ánh sáng, nhiệt độ,...
   RUNG wire#powerrail
      "CONDITION"(SIM_MODE := "SIM_MODE", MW_ANH_SANG := "MW_ANH_SANG", MW_DO_AM := "MW_DO_AM", MW_NHIET_DO := "MW_NHIET_DO", MW_DO_AM_DAT := "MW_DO_AM_DAT", IW_ANH_SANG => "IW_ANH_SANG", IW_DO_AM => "IW_DO_AM", IW_NHIET_DO => "IW_NHIET_DO", IW_DO_AM_DAT => "IW_DO_AM_DAT")
   END_RUNG
   // the same network as SCL:
   "CONDITION"(SIM_MODE := "SIM_MODE",
               MW_ANH_SANG := "MW_ANH_SANG",
               MW_DO_AM := "MW_DO_AM",
               MW_NHIET_DO := "MW_NHIET_DO",
               MW_DO_AM_DAT := "MW_DO_AM_DAT",
               IW_ANH_SANG => "IW_ANH_SANG",
               IW_DO_AM => "IW_DO_AM",
               IW_NHIET_DO => "IW_NHIET_DO",
               IW_DO_AM_DAT => "IW_DO_AM_DAT");
END_REGION

REGION Network 4
   RUNG wire#powerrail
      "SIMULATE"()
   END_RUNG
   // the same network as SCL:
   "SIMULATE"();
END_REGION

REGION Network 5: Chuyển đổi giá trị Analog sang dạng số
   // ENO of a box is taken as its EN; it also drops when the box reports an error
   "RET_VAL1" := SCALE(IN := "IW_NHIET_DO",
                       HI_LIM := 100.0,
                       LO_LIM := 0.0,
                       BIPOLAR := "BIPOLAR",
                       OUT => "TT_NHIET_DO");
   "RET_VAL2" := SCALE(IN := "IW_DO_AM_DAT",
                       HI_LIM := 100.0,
                       LO_LIM := 0.0,
                       BIPOLAR := "BIPOLAR",
                       OUT => "TT_DO_AM_DAT");
END_REGION

REGION Network 6
   // ENO of a box is taken as its EN; it also drops when the box reports an error
   "RET_VAL3" := SCALE(IN := "IW_DO_AM",
                       HI_LIM := 100.0,
                       LO_LIM := 0.0,
                       BIPOLAR := "BIPOLAR",
                       OUT => "TT_DO_AM");
   "RET_VAL4" := SCALE(IN := "IW_ANH_SANG",
                       HI_LIM := 100.0,
                       LO_LIM := 0.0,
                       BIPOLAR := "BIPOLAR",
                       OUT => "TT_ANH_SANG");
END_REGION

REGION Network 7: Đọc thời gian hệ thống
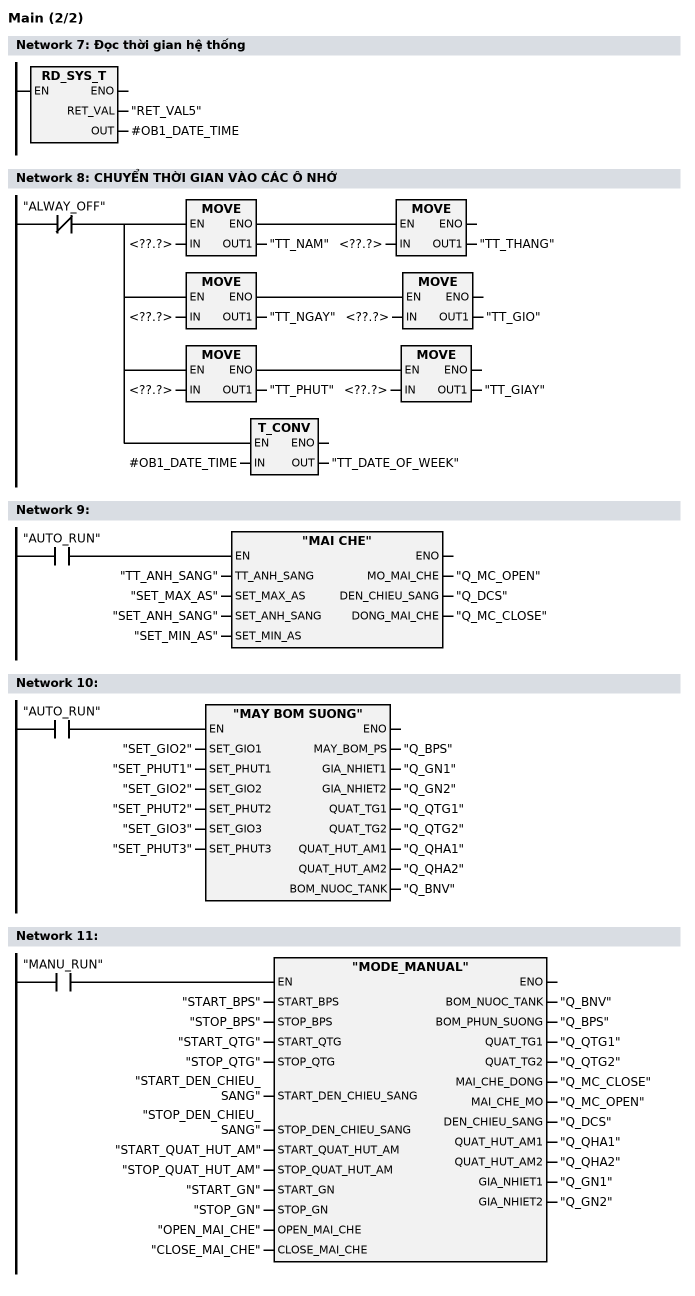
   "RET_VAL5" := RD_SYS_T(OUT => #OB1_DATE_TIME);
END_REGION

REGION Network 8: CHUYỂN THỜI GIAN VÀO CÁC Ô NHỚ
   // ENO of a box is taken as its EN; it also drops when the box reports an error
   IF NOT "ALWAY_OFF" THEN
       "TT_NAM" := <??.?>;
       "TT_THANG" := <??.?>;
       "TT_NGAY" := <??.?>;
       "TT_GIO" := <??.?>;
       "TT_PHUT" := <??.?>;
       "TT_GIAY" := <??.?>;
       "TT_DATE_OF_WEEK" := T_CONV(IN := #OB1_DATE_TIME);
   END_IF;
END_REGION

REGION Network 9
   RUNG wire#powerrail
      Contact( "AUTO_RUN" )
      "MAI CHE"(TT_ANH_SANG := "TT_ANH_SANG", SET_MAX_AS := "SET_MAX_AS", SET_ANH_SANG := "SET_ANH_SANG", SET_MIN_AS := "SET_MIN_AS", MO_MAI_CHE => "Q_MC_OPEN", DEN_CHIEU_SANG => "Q_DCS", DONG_MAI_CHE => "Q_MC_CLOSE")
   END_RUNG
   // the same network as SCL:
   IF "AUTO_RUN" THEN
       "MAI CHE"(TT_ANH_SANG := "TT_ANH_SANG",
                 SET_MAX_AS := "SET_MAX_AS",
                 SET_ANH_SANG := "SET_ANH_SANG",
                 SET_MIN_AS := "SET_MIN_AS",
                 MO_MAI_CHE => "Q_MC_OPEN",
                 DEN_CHIEU_SANG => "Q_DCS",
                 DONG_MAI_CHE => "Q_MC_CLOSE");
   END_IF;
END_REGION

REGION Network 10
   RUNG wire#powerrail
      Contact( "AUTO_RUN" )
      "MAY BOM SUONG"(SET_GIO1 := "SET_GIO2", SET_PHUT1 := "SET_PHUT1", SET_GIO2 := "SET_GIO2", SET_PHUT2 := "SET_PHUT2", SET_GIO3 := "SET_GIO3", SET_PHUT3 := "SET_PHUT3", MAY_BOM_PS => "Q_BPS", GIA_NHIET1 => "Q_GN1", GIA_NHIET2 => "Q_GN2", QUAT_TG1 => "Q_QTG1", QUAT_TG2 => "Q_QTG2", QUAT_HUT_AM1 => "Q_QHA1", QUAT_HUT_AM2 => "Q_QHA2", BOM_NUOC_TANK => "Q_BNV")
   END_RUNG
   // the same network as SCL:
   IF "AUTO_RUN" THEN
       "MAY BOM SUONG"(SET_GIO1 := "SET_GIO2",
                       SET_PHUT1 := "SET_PHUT1",
                       SET_GIO2 := "SET_GIO2",
                       SET_PHUT2 := "SET_PHUT2",
                       SET_GIO3 := "SET_GIO3",
                       SET_PHUT3 := "SET_PHUT3",
                       MAY_BOM_PS => "Q_BPS",
                       GIA_NHIET1 => "Q_GN1",
                       GIA_NHIET2 => "Q_GN2",
                       QUAT_TG1 => "Q_QTG1",
                       QUAT_TG2 => "Q_QTG2",
                       QUAT_HUT_AM1 => "Q_QHA1",
                       QUAT_HUT_AM2 => "Q_QHA2",
                       BOM_NUOC_TANK => "Q_BNV");
   END_IF;
END_REGION

REGION Network 11
   RUNG wire#powerrail
      Contact( "MANU_RUN" )
      "MODE_MANUAL"(START_BPS := "START_BPS", STOP_BPS := "STOP_BPS", START_QTG := "START_QTG", STOP_QTG := "STOP_QTG", START_DEN_CHIEU_SANG := "START_DEN_CHIEU_SANG", STOP_DEN_CHIEU_SANG := "STOP_DEN_CHIEU_SANG", START_QUAT_HUT_AM := "START_QUAT_HUT_AM", STOP_QUAT_HUT_AM := "STOP_QUAT_HUT_AM", START_GN := "START_GN", STOP_GN := "STOP_GN", OPEN_MAI_CHE := "OPEN_MAI_CHE", CLOSE_MAI_CHE := "CLOSE_MAI_CHE", BOM_NUOC_TANK => "Q_BNV", BOM_PHUN_SUONG => "Q_BPS", QUAT_TG1 => "Q_QTG1", QUAT_TG2 => "Q_QTG2", MAI_CHE_DONG => "Q_MC_CLOSE", MAI_CHE_MO => "Q_MC_OPEN", DEN_CHIEU_SANG => "Q_DCS", QUAT_HUT_AM1 => "Q_QHA1", QUAT_HUT_AM2 => "Q_QHA2", GIA_NHIET1 => "Q_GN1", GIA_NHIET2 => "Q_GN2")
   END_RUNG
   // the same network as SCL:
   IF "MANU_RUN" THEN
       "MODE_MANUAL"(START_BPS := "START_BPS",
                     STOP_BPS := "STOP_BPS",
                     START_QTG := "START_QTG",
                     STOP_QTG := "STOP_QTG",
                     START_DEN_CHIEU_SANG := "START_DEN_CHIEU_SANG",
                     STOP_DEN_CHIEU_SANG := "STOP_DEN_CHIEU_SANG",
                     START_QUAT_HUT_AM := "START_QUAT_HUT_AM",
                     STOP_QUAT_HUT_AM := "STOP_QUAT_HUT_AM",
                     START_GN := "START_GN",
                     STOP_GN := "STOP_GN",
                     OPEN_MAI_CHE := "OPEN_MAI_CHE",
                     CLOSE_MAI_CHE := "CLOSE_MAI_CHE",
                     BOM_NUOC_TANK => "Q_BNV",
                     BOM_PHUN_SUONG => "Q_BPS",
                     QUAT_TG1 => "Q_QTG1",
                     QUAT_TG2 => "Q_QTG2",
                     MAI_CHE_DONG => "Q_MC_CLOSE",
                     MAI_CHE_MO => "Q_MC_OPEN",
                     DEN_CHIEU_SANG => "Q_DCS",
                     QUAT_HUT_AM1 => "Q_QHA1",
                     QUAT_HUT_AM2 => "Q_QHA2",
                     GIA_NHIET1 => "Q_GN1",
                     GIA_NHIET2 => "Q_GN2");
   END_IF;
END_REGION
END_ORGANIZATION_BLOCK